# EPICS substitutions: modules/event/evrIoc/Db/evrPatternXL16.substitutions
#
# Pattern records
file evrPatternAll.db
{
#	    Device        ,SLC Pattern  EVR/Trigger
#	                   Check LNK      Links
  pattern { DEVICE        ,  LINK4    , LINK5, LINK6, TREF   , TS1ST, TS2ND}
	  { IOC:XL16:EV01 ,   ""      ,  ""  ,  ""  , 1.03E06,   1  ,   4  }
}
# Event records
file evrEventAll.db
{
  pattern { DEVICE   , TREF }
	  { IOC:XL16:EV01, 1E06 }
}
